{attribute 'Tc2GvlVarNames'}
VAR_GLOBAL CONSTANT
	(* Regelung_Modus Heizstäbe *)
	E_HS_Regelung_Modus_Default_unten	: SINT := 0;
	E_HS_Regelung_Modus_oben			: SINT := 1;
	E_HS_Regelung_Modus_mitte			: SINT := 2;
	E_HS_Regelung_Modus_unten			: SINT := 3;
END_VAR

(* stored: Version 1.1.0.1, ProductVersion 3.1.4024.9
   GVL Con_HS: Id {9ae17114-8102-4bbf-a468-f9822b569210} *)
